// TIA Portal V17 export
// export: Created 2022-03-12T16:05:14.101526Z, ExportSetting WithDefaults, DisplayName Totally Integrated Automation Portal, DisplayVersion V17, DisplayName TIA Portal Openness, DisplayVersion V17, DisplayName TIA Portal Version Control Interface, DisplayVersion V17, DisplayName STEP 7 Professional, DisplayVersion V17, DisplayName STEP 7 Safety, DisplayVersion V17, DisplayName WinCC Advanced / Unified PC, DisplayVersion V17
FUNCTION_BLOCK "UN_01_PackML_ModuleSum"   // FB31621, LAD
TITLE = UN_01_PackML_ModuleSummation
{ S7_Optimized_Access := 'TRUE' }
AUTHOR : tech.team.motioncontrol@siemens.com
FAMILY : CPG
VERSION : 1.0
// Support: tech.team.motioncontrol@siemens.com
// Fax: +49 (0) 9131/98-1297
// stored: AutoNumber true, IsIECCheckEnabled false, IsRetainMemResEnabled false, MemoryReserve 100, SetENOAutomatically false, UDAEnableTagReadback false
   VAR
      statDummyBool { ExternalAccessible := 'False'; ExternalVisible := 'False'; ExternalWritable := 'False'} : Bool;   // dummy bool - placeholder
   END_VAR
BEGIN

REGION Network 1: UN - Reset Command
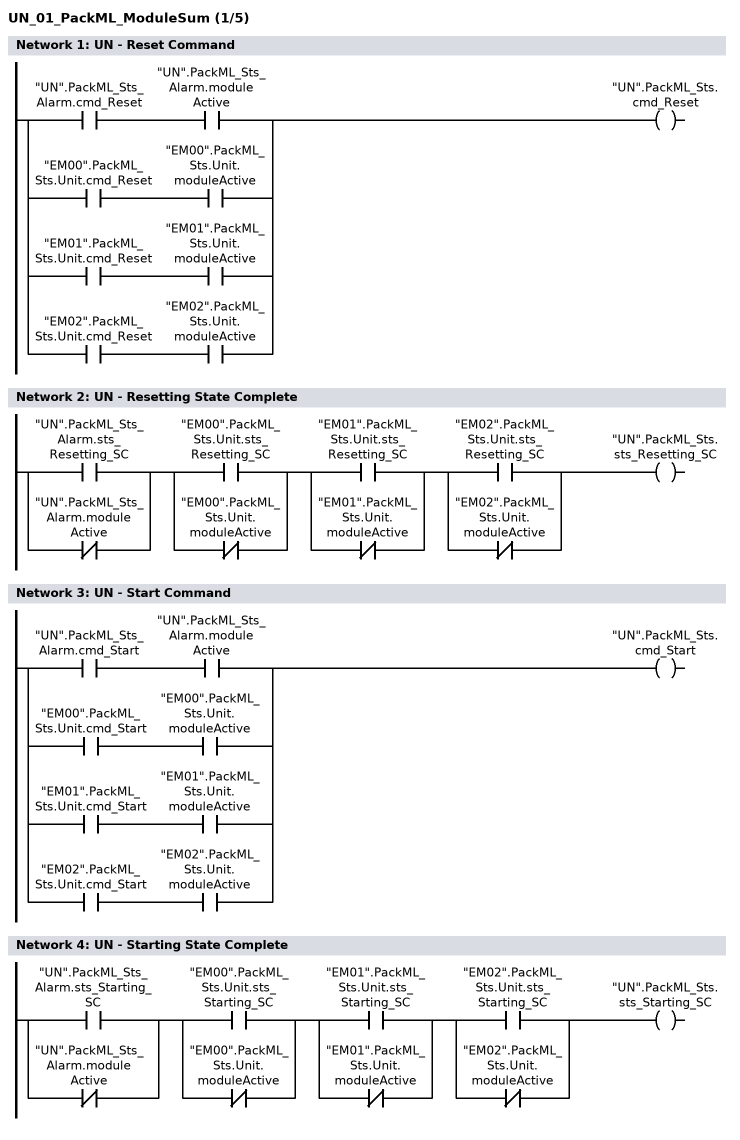
   RUNG wire#powerrail
      Contact( "UN".PackML_Sts_Alarm.cmd_Reset )
      Contact( "UN".PackML_Sts_Alarm.moduleActive )
      wire#w1
      Coil( "UN".PackML_Sts.cmd_Reset )
   END_RUNG
   RUNG wire#powerrail
      Contact( "EM00".PackML_Sts.Unit.cmd_Reset )
      Contact( "EM00".PackML_Sts.Unit.moduleActive )
   END_RUNG wire#w1
   RUNG wire#powerrail
      Contact( "EM01".PackML_Sts.Unit.cmd_Reset )
      Contact( "EM01".PackML_Sts.Unit.moduleActive )
   END_RUNG wire#w1
   RUNG wire#powerrail
      Contact( "EM02".PackML_Sts.Unit.cmd_Reset )
      Contact( "EM02".PackML_Sts.Unit.moduleActive )
   END_RUNG wire#w1
   // the same network as SCL:
   "UN".PackML_Sts.cmd_Reset := ("UN".PackML_Sts_Alarm.cmd_Reset AND "UN".PackML_Sts_Alarm.moduleActive) OR ("EM00".PackML_Sts.Unit.cmd_Reset AND "EM00".PackML_Sts.Unit.moduleActive) OR ("EM01".PackML_Sts.Unit.cmd_Reset AND "EM01".PackML_Sts.Unit.moduleActive) OR ("EM02".PackML_Sts.Unit.cmd_Reset AND "EM02".PackML_Sts.Unit.moduleActive);
END_REGION

REGION Network 2: UN - Resetting State Complete
   RUNG wire#powerrail
      Contact( "UN".PackML_Sts_Alarm.sts_Resetting_SC )
      wire#w1
      Contact( "EM00".PackML_Sts.Unit.sts_Resetting_SC )
      wire#w2
      Contact( "EM01".PackML_Sts.Unit.sts_Resetting_SC )
      wire#w3
      Contact( "EM02".PackML_Sts.Unit.sts_Resetting_SC )
      wire#w4
      Coil( "UN".PackML_Sts.sts_Resetting_SC )
   END_RUNG
   RUNG wire#powerrail
      I_Contact( "UN".PackML_Sts_Alarm.moduleActive )
   END_RUNG wire#w1
   RUNG wire#w1
      I_Contact( "EM00".PackML_Sts.Unit.moduleActive )
   END_RUNG wire#w2
   RUNG wire#w2
      I_Contact( "EM01".PackML_Sts.Unit.moduleActive )
   END_RUNG wire#w3
   RUNG wire#w3
      I_Contact( "EM02".PackML_Sts.Unit.moduleActive )
   END_RUNG wire#w4
   // the same network as SCL:
   "UN".PackML_Sts.sts_Resetting_SC := ("UN".PackML_Sts_Alarm.sts_Resetting_SC OR NOT "UN".PackML_Sts_Alarm.moduleActive) AND ("EM00".PackML_Sts.Unit.sts_Resetting_SC OR NOT "EM00".PackML_Sts.Unit.moduleActive) AND ("EM01".PackML_Sts.Unit.sts_Resetting_SC OR NOT "EM01".PackML_Sts.Unit.moduleActive) AND ("EM02".PackML_Sts.Unit.sts_Resetting_SC OR NOT "EM02".PackML_Sts.Unit.moduleActive);
END_REGION

REGION Network 3: UN - Start Command
   RUNG wire#powerrail
      Contact( "UN".PackML_Sts_Alarm.cmd_Start )
      Contact( "UN".PackML_Sts_Alarm.moduleActive )
      wire#w1
      Coil( "UN".PackML_Sts.cmd_Start )
   END_RUNG
   RUNG wire#powerrail
      Contact( "EM00".PackML_Sts.Unit.cmd_Start )
      Contact( "EM00".PackML_Sts.Unit.moduleActive )
   END_RUNG wire#w1
   RUNG wire#powerrail
      Contact( "EM01".PackML_Sts.Unit.cmd_Start )
      Contact( "EM01".PackML_Sts.Unit.moduleActive )
   END_RUNG wire#w1
   RUNG wire#powerrail
      Contact( "EM02".PackML_Sts.Unit.cmd_Start )
      Contact( "EM02".PackML_Sts.Unit.moduleActive )
   END_RUNG wire#w1
   // the same network as SCL:
   "UN".PackML_Sts.cmd_Start := ("UN".PackML_Sts_Alarm.cmd_Start AND "UN".PackML_Sts_Alarm.moduleActive) OR ("EM00".PackML_Sts.Unit.cmd_Start AND "EM00".PackML_Sts.Unit.moduleActive) OR ("EM01".PackML_Sts.Unit.cmd_Start AND "EM01".PackML_Sts.Unit.moduleActive) OR ("EM02".PackML_Sts.Unit.cmd_Start AND "EM02".PackML_Sts.Unit.moduleActive);
END_REGION

REGION Network 4: UN - Starting State Complete
   RUNG wire#powerrail
      Contact( "UN".PackML_Sts_Alarm.sts_Starting_SC )
      wire#w1
      Contact( "EM00".PackML_Sts.Unit.sts_Starting_SC )
      wire#w2
      Contact( "EM01".PackML_Sts.Unit.sts_Starting_SC )
      wire#w3
      Contact( "EM02".PackML_Sts.Unit.sts_Starting_SC )
      wire#w4
      Coil( "UN".PackML_Sts.sts_Starting_SC )
   END_RUNG
   RUNG wire#powerrail
      I_Contact( "UN".PackML_Sts_Alarm.moduleActive )
   END_RUNG wire#w1
   RUNG wire#w1
      I_Contact( "EM00".PackML_Sts.Unit.moduleActive )
   END_RUNG wire#w2
   RUNG wire#w2
      I_Contact( "EM01".PackML_Sts.Unit.moduleActive )
   END_RUNG wire#w3
   RUNG wire#w3
      I_Contact( "EM02".PackML_Sts.Unit.moduleActive )
   END_RUNG wire#w4
   // the same network as SCL:
   "UN".PackML_Sts.sts_Starting_SC := ("UN".PackML_Sts_Alarm.sts_Starting_SC OR NOT "UN".PackML_Sts_Alarm.moduleActive) AND ("EM00".PackML_Sts.Unit.sts_Starting_SC OR NOT "EM00".PackML_Sts.Unit.moduleActive) AND ("EM01".PackML_Sts.Unit.sts_Starting_SC OR NOT "EM01".PackML_Sts.Unit.moduleActive) AND ("EM02".PackML_Sts.Unit.sts_Starting_SC OR NOT "EM02".PackML_Sts.Unit.moduleActive);
END_REGION

REGION Network 5: UN - Stop Command
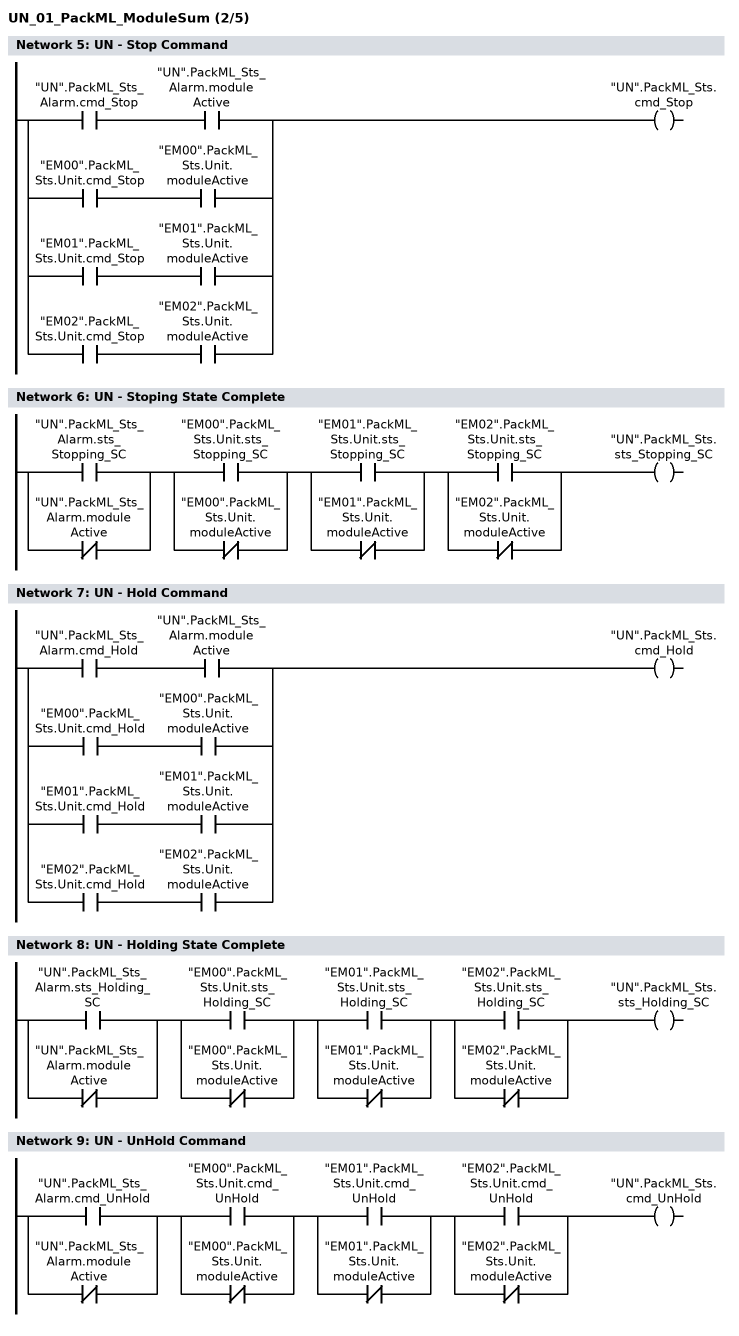
   RUNG wire#powerrail
      Contact( "UN".PackML_Sts_Alarm.cmd_Stop )
      Contact( "UN".PackML_Sts_Alarm.moduleActive )
      wire#w1
      Coil( "UN".PackML_Sts.cmd_Stop )
   END_RUNG
   RUNG wire#powerrail
      Contact( "EM00".PackML_Sts.Unit.cmd_Stop )
      Contact( "EM00".PackML_Sts.Unit.moduleActive )
   END_RUNG wire#w1
   RUNG wire#powerrail
      Contact( "EM01".PackML_Sts.Unit.cmd_Stop )
      Contact( "EM01".PackML_Sts.Unit.moduleActive )
   END_RUNG wire#w1
   RUNG wire#powerrail
      Contact( "EM02".PackML_Sts.Unit.cmd_Stop )
      Contact( "EM02".PackML_Sts.Unit.moduleActive )
   END_RUNG wire#w1
   // the same network as SCL:
   "UN".PackML_Sts.cmd_Stop := ("UN".PackML_Sts_Alarm.cmd_Stop AND "UN".PackML_Sts_Alarm.moduleActive) OR ("EM00".PackML_Sts.Unit.cmd_Stop AND "EM00".PackML_Sts.Unit.moduleActive) OR ("EM01".PackML_Sts.Unit.cmd_Stop AND "EM01".PackML_Sts.Unit.moduleActive) OR ("EM02".PackML_Sts.Unit.cmd_Stop AND "EM02".PackML_Sts.Unit.moduleActive);
END_REGION

REGION Network 6: UN - Stoping State Complete
   RUNG wire#powerrail
      Contact( "UN".PackML_Sts_Alarm.sts_Stopping_SC )
      wire#w1
      Contact( "EM00".PackML_Sts.Unit.sts_Stopping_SC )
      wire#w2
      Contact( "EM01".PackML_Sts.Unit.sts_Stopping_SC )
      wire#w3
      Contact( "EM02".PackML_Sts.Unit.sts_Stopping_SC )
      wire#w4
      Coil( "UN".PackML_Sts.sts_Stopping_SC )
   END_RUNG
   RUNG wire#powerrail
      I_Contact( "UN".PackML_Sts_Alarm.moduleActive )
   END_RUNG wire#w1
   RUNG wire#w1
      I_Contact( "EM00".PackML_Sts.Unit.moduleActive )
   END_RUNG wire#w2
   RUNG wire#w2
      I_Contact( "EM01".PackML_Sts.Unit.moduleActive )
   END_RUNG wire#w3
   RUNG wire#w3
      I_Contact( "EM02".PackML_Sts.Unit.moduleActive )
   END_RUNG wire#w4
   // the same network as SCL:
   "UN".PackML_Sts.sts_Stopping_SC := ("UN".PackML_Sts_Alarm.sts_Stopping_SC OR NOT "UN".PackML_Sts_Alarm.moduleActive) AND ("EM00".PackML_Sts.Unit.sts_Stopping_SC OR NOT "EM00".PackML_Sts.Unit.moduleActive) AND ("EM01".PackML_Sts.Unit.sts_Stopping_SC OR NOT "EM01".PackML_Sts.Unit.moduleActive) AND ("EM02".PackML_Sts.Unit.sts_Stopping_SC OR NOT "EM02".PackML_Sts.Unit.moduleActive);
END_REGION

REGION Network 7: UN - Hold Command
   RUNG wire#powerrail
      Contact( "UN".PackML_Sts_Alarm.cmd_Hold )
      Contact( "UN".PackML_Sts_Alarm.moduleActive )
      wire#w1
      Coil( "UN".PackML_Sts.cmd_Hold )
   END_RUNG
   RUNG wire#powerrail
      Contact( "EM00".PackML_Sts.Unit.cmd_Hold )
      Contact( "EM00".PackML_Sts.Unit.moduleActive )
   END_RUNG wire#w1
   RUNG wire#powerrail
      Contact( "EM01".PackML_Sts.Unit.cmd_Hold )
      Contact( "EM01".PackML_Sts.Unit.moduleActive )
   END_RUNG wire#w1
   RUNG wire#powerrail
      Contact( "EM02".PackML_Sts.Unit.cmd_Hold )
      Contact( "EM02".PackML_Sts.Unit.moduleActive )
   END_RUNG wire#w1
   // the same network as SCL:
   "UN".PackML_Sts.cmd_Hold := ("UN".PackML_Sts_Alarm.cmd_Hold AND "UN".PackML_Sts_Alarm.moduleActive) OR ("EM00".PackML_Sts.Unit.cmd_Hold AND "EM00".PackML_Sts.Unit.moduleActive) OR ("EM01".PackML_Sts.Unit.cmd_Hold AND "EM01".PackML_Sts.Unit.moduleActive) OR ("EM02".PackML_Sts.Unit.cmd_Hold AND "EM02".PackML_Sts.Unit.moduleActive);
END_REGION

REGION Network 8: UN - Holding State Complete
   RUNG wire#powerrail
      Contact( "UN".PackML_Sts_Alarm.sts_Holding_SC )
      wire#w1
      Contact( "EM00".PackML_Sts.Unit.sts_Holding_SC )
      wire#w2
      Contact( "EM01".PackML_Sts.Unit.sts_Holding_SC )
      wire#w3
      Contact( "EM02".PackML_Sts.Unit.sts_Holding_SC )
      wire#w4
      Coil( "UN".PackML_Sts.sts_Holding_SC )
   END_RUNG
   RUNG wire#powerrail
      I_Contact( "UN".PackML_Sts_Alarm.moduleActive )
   END_RUNG wire#w1
   RUNG wire#w1
      I_Contact( "EM00".PackML_Sts.Unit.moduleActive )
   END_RUNG wire#w2
   RUNG wire#w2
      I_Contact( "EM01".PackML_Sts.Unit.moduleActive )
   END_RUNG wire#w3
   RUNG wire#w3
      I_Contact( "EM02".PackML_Sts.Unit.moduleActive )
   END_RUNG wire#w4
   // the same network as SCL:
   "UN".PackML_Sts.sts_Holding_SC := ("UN".PackML_Sts_Alarm.sts_Holding_SC OR NOT "UN".PackML_Sts_Alarm.moduleActive) AND ("EM00".PackML_Sts.Unit.sts_Holding_SC OR NOT "EM00".PackML_Sts.Unit.moduleActive) AND ("EM01".PackML_Sts.Unit.sts_Holding_SC OR NOT "EM01".PackML_Sts.Unit.moduleActive) AND ("EM02".PackML_Sts.Unit.sts_Holding_SC OR NOT "EM02".PackML_Sts.Unit.moduleActive);
END_REGION

REGION Network 9: UN - UnHold Command
   RUNG wire#powerrail
      Contact( "UN".PackML_Sts_Alarm.cmd_UnHold )
      wire#w1
      Contact( "EM00".PackML_Sts.Unit.cmd_UnHold )
      wire#w2
      Contact( "EM01".PackML_Sts.Unit.cmd_UnHold )
      wire#w3
      Contact( "EM02".PackML_Sts.Unit.cmd_UnHold )
      wire#w4
      Coil( "UN".PackML_Sts.cmd_UnHold )
   END_RUNG
   RUNG wire#powerrail
      I_Contact( "UN".PackML_Sts_Alarm.moduleActive )
   END_RUNG wire#w1
   RUNG wire#w1
      I_Contact( "EM00".PackML_Sts.Unit.moduleActive )
   END_RUNG wire#w2
   RUNG wire#w2
      I_Contact( "EM01".PackML_Sts.Unit.moduleActive )
   END_RUNG wire#w3
   RUNG wire#w3
      I_Contact( "EM02".PackML_Sts.Unit.moduleActive )
   END_RUNG wire#w4
   // the same network as SCL:
   "UN".PackML_Sts.cmd_UnHold := ("UN".PackML_Sts_Alarm.cmd_UnHold OR NOT "UN".PackML_Sts_Alarm.moduleActive) AND ("EM00".PackML_Sts.Unit.cmd_UnHold OR NOT "EM00".PackML_Sts.Unit.moduleActive) AND ("EM01".PackML_Sts.Unit.cmd_UnHold OR NOT "EM01".PackML_Sts.Unit.moduleActive) AND ("EM02".PackML_Sts.Unit.cmd_UnHold OR NOT "EM02".PackML_Sts.Unit.moduleActive);
END_REGION

REGION Network 10: UN - UnHolding State Complete
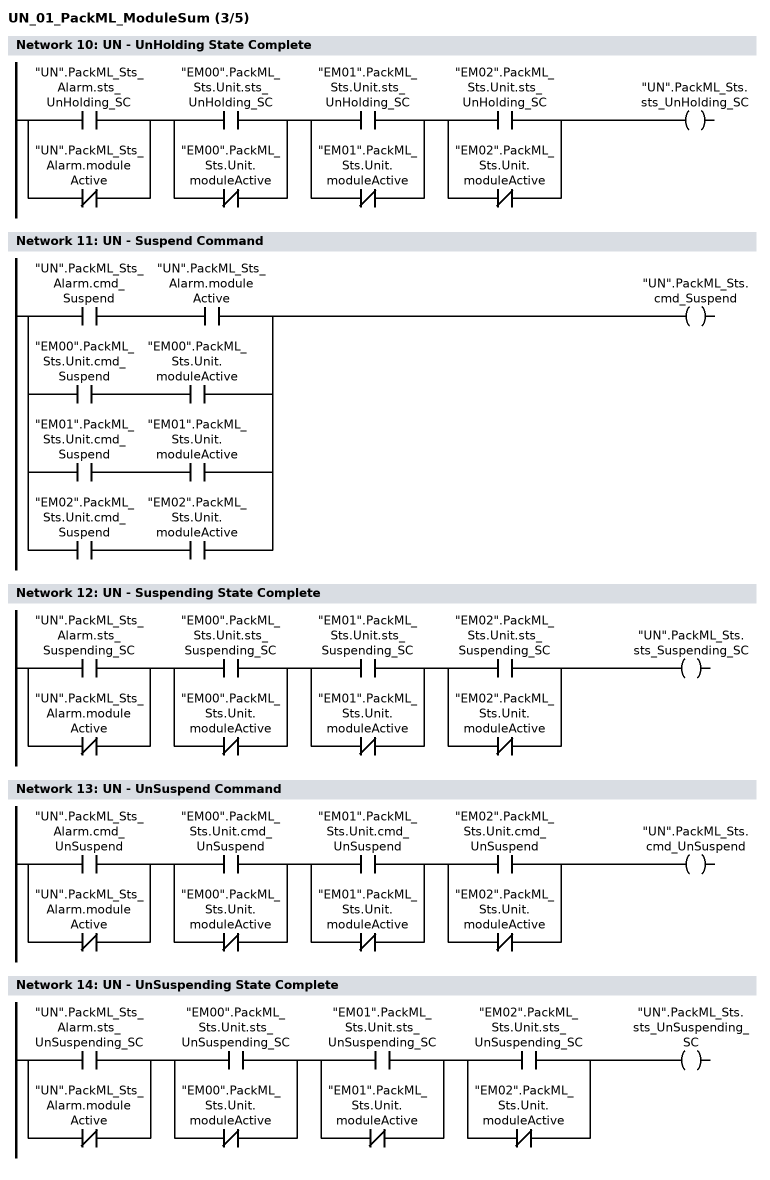
   RUNG wire#powerrail
      Contact( "UN".PackML_Sts_Alarm.sts_UnHolding_SC )
      wire#w1
      Contact( "EM00".PackML_Sts.Unit.sts_UnHolding_SC )
      wire#w2
      Contact( "EM01".PackML_Sts.Unit.sts_UnHolding_SC )
      wire#w3
      Contact( "EM02".PackML_Sts.Unit.sts_UnHolding_SC )
      wire#w4
      Coil( "UN".PackML_Sts.sts_UnHolding_SC )
   END_RUNG
   RUNG wire#powerrail
      I_Contact( "UN".PackML_Sts_Alarm.moduleActive )
   END_RUNG wire#w1
   RUNG wire#w1
      I_Contact( "EM00".PackML_Sts.Unit.moduleActive )
   END_RUNG wire#w2
   RUNG wire#w2
      I_Contact( "EM01".PackML_Sts.Unit.moduleActive )
   END_RUNG wire#w3
   RUNG wire#w3
      I_Contact( "EM02".PackML_Sts.Unit.moduleActive )
   END_RUNG wire#w4
   // the same network as SCL:
   "UN".PackML_Sts.sts_UnHolding_SC := ("UN".PackML_Sts_Alarm.sts_UnHolding_SC OR NOT "UN".PackML_Sts_Alarm.moduleActive) AND ("EM00".PackML_Sts.Unit.sts_UnHolding_SC OR NOT "EM00".PackML_Sts.Unit.moduleActive) AND ("EM01".PackML_Sts.Unit.sts_UnHolding_SC OR NOT "EM01".PackML_Sts.Unit.moduleActive) AND ("EM02".PackML_Sts.Unit.sts_UnHolding_SC OR NOT "EM02".PackML_Sts.Unit.moduleActive);
END_REGION

REGION Network 11: UN - Suspend Command
   RUNG wire#powerrail
      Contact( "UN".PackML_Sts_Alarm.cmd_Suspend )
      Contact( "UN".PackML_Sts_Alarm.moduleActive )
      wire#w1
      Coil( "UN".PackML_Sts.cmd_Suspend )
   END_RUNG
   RUNG wire#powerrail
      Contact( "EM00".PackML_Sts.Unit.cmd_Suspend )
      Contact( "EM00".PackML_Sts.Unit.moduleActive )
   END_RUNG wire#w1
   RUNG wire#powerrail
      Contact( "EM01".PackML_Sts.Unit.cmd_Suspend )
      Contact( "EM01".PackML_Sts.Unit.moduleActive )
   END_RUNG wire#w1
   RUNG wire#powerrail
      Contact( "EM02".PackML_Sts.Unit.cmd_Suspend )
      Contact( "EM02".PackML_Sts.Unit.moduleActive )
   END_RUNG wire#w1
   // the same network as SCL:
   "UN".PackML_Sts.cmd_Suspend := ("UN".PackML_Sts_Alarm.cmd_Suspend AND "UN".PackML_Sts_Alarm.moduleActive) OR ("EM00".PackML_Sts.Unit.cmd_Suspend AND "EM00".PackML_Sts.Unit.moduleActive) OR ("EM01".PackML_Sts.Unit.cmd_Suspend AND "EM01".PackML_Sts.Unit.moduleActive) OR ("EM02".PackML_Sts.Unit.cmd_Suspend AND "EM02".PackML_Sts.Unit.moduleActive);
END_REGION

REGION Network 12: UN - Suspending State Complete
   RUNG wire#powerrail
      Contact( "UN".PackML_Sts_Alarm.sts_Suspending_SC )
      wire#w1
      Contact( "EM00".PackML_Sts.Unit.sts_Suspending_SC )
      wire#w2
      Contact( "EM01".PackML_Sts.Unit.sts_Suspending_SC )
      wire#w3
      Contact( "EM02".PackML_Sts.Unit.sts_Suspending_SC )
      wire#w4
      Coil( "UN".PackML_Sts.sts_Suspending_SC )
   END_RUNG
   RUNG wire#powerrail
      I_Contact( "UN".PackML_Sts_Alarm.moduleActive )
   END_RUNG wire#w1
   RUNG wire#w1
      I_Contact( "EM00".PackML_Sts.Unit.moduleActive )
   END_RUNG wire#w2
   RUNG wire#w2
      I_Contact( "EM01".PackML_Sts.Unit.moduleActive )
   END_RUNG wire#w3
   RUNG wire#w3
      I_Contact( "EM02".PackML_Sts.Unit.moduleActive )
   END_RUNG wire#w4
   // the same network as SCL:
   "UN".PackML_Sts.sts_Suspending_SC := ("UN".PackML_Sts_Alarm.sts_Suspending_SC OR NOT "UN".PackML_Sts_Alarm.moduleActive) AND ("EM00".PackML_Sts.Unit.sts_Suspending_SC OR NOT "EM00".PackML_Sts.Unit.moduleActive) AND ("EM01".PackML_Sts.Unit.sts_Suspending_SC OR NOT "EM01".PackML_Sts.Unit.moduleActive) AND ("EM02".PackML_Sts.Unit.sts_Suspending_SC OR NOT "EM02".PackML_Sts.Unit.moduleActive);
END_REGION

REGION Network 13: UN - UnSuspend Command
   RUNG wire#powerrail
      Contact( "UN".PackML_Sts_Alarm.cmd_UnSuspend )
      wire#w1
      Contact( "EM00".PackML_Sts.Unit.cmd_UnSuspend )
      wire#w2
      Contact( "EM01".PackML_Sts.Unit.cmd_UnSuspend )
      wire#w3
      Contact( "EM02".PackML_Sts.Unit.cmd_UnSuspend )
      wire#w4
      Coil( "UN".PackML_Sts.cmd_UnSuspend )
   END_RUNG
   RUNG wire#powerrail
      I_Contact( "UN".PackML_Sts_Alarm.moduleActive )
   END_RUNG wire#w1
   RUNG wire#w1
      I_Contact( "EM00".PackML_Sts.Unit.moduleActive )
   END_RUNG wire#w2
   RUNG wire#w2
      I_Contact( "EM01".PackML_Sts.Unit.moduleActive )
   END_RUNG wire#w3
   RUNG wire#w3
      I_Contact( "EM02".PackML_Sts.Unit.moduleActive )
   END_RUNG wire#w4
   // the same network as SCL:
   "UN".PackML_Sts.cmd_UnSuspend := ("UN".PackML_Sts_Alarm.cmd_UnSuspend OR NOT "UN".PackML_Sts_Alarm.moduleActive) AND ("EM00".PackML_Sts.Unit.cmd_UnSuspend OR NOT "EM00".PackML_Sts.Unit.moduleActive) AND ("EM01".PackML_Sts.Unit.cmd_UnSuspend OR NOT "EM01".PackML_Sts.Unit.moduleActive) AND ("EM02".PackML_Sts.Unit.cmd_UnSuspend OR NOT "EM02".PackML_Sts.Unit.moduleActive);
END_REGION

REGION Network 14: UN - UnSuspending State Complete
   RUNG wire#powerrail
      Contact( "UN".PackML_Sts_Alarm.sts_UnSuspending_SC )
      wire#w1
      Contact( "EM00".PackML_Sts.Unit.sts_UnSuspending_SC )
      wire#w2
      Contact( "EM01".PackML_Sts.Unit.sts_UnSuspending_SC )
      wire#w3
      Contact( "EM02".PackML_Sts.Unit.sts_UnSuspending_SC )
      wire#w4
      Coil( "UN".PackML_Sts.sts_UnSuspending_SC )
   END_RUNG
   RUNG wire#powerrail
      I_Contact( "UN".PackML_Sts_Alarm.moduleActive )
   END_RUNG wire#w1
   RUNG wire#w1
      I_Contact( "EM00".PackML_Sts.Unit.moduleActive )
   END_RUNG wire#w2
   RUNG wire#w2
      I_Contact( "EM01".PackML_Sts.Unit.moduleActive )
   END_RUNG wire#w3
   RUNG wire#w3
      I_Contact( "EM02".PackML_Sts.Unit.moduleActive )
   END_RUNG wire#w4
   // the same network as SCL:
   "UN".PackML_Sts.sts_UnSuspending_SC := ("UN".PackML_Sts_Alarm.sts_UnSuspending_SC OR NOT "UN".PackML_Sts_Alarm.moduleActive) AND ("EM00".PackML_Sts.Unit.sts_UnSuspending_SC OR NOT "EM00".PackML_Sts.Unit.moduleActive) AND ("EM01".PackML_Sts.Unit.sts_UnSuspending_SC OR NOT "EM01".PackML_Sts.Unit.moduleActive) AND ("EM02".PackML_Sts.Unit.sts_UnSuspending_SC OR NOT "EM02".PackML_Sts.Unit.moduleActive);
END_REGION

REGION Network 15: UN - Abort Command
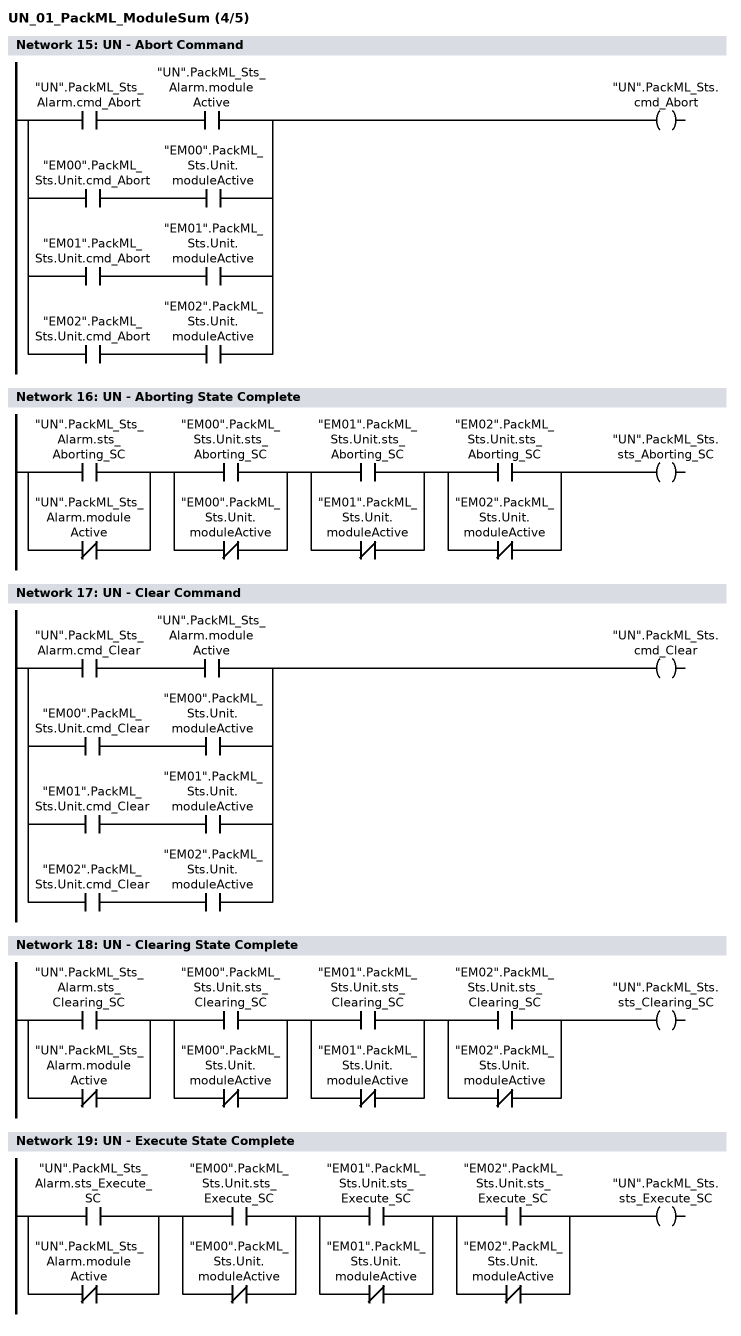
   RUNG wire#powerrail
      Contact( "UN".PackML_Sts_Alarm.cmd_Abort )
      Contact( "UN".PackML_Sts_Alarm.moduleActive )
      wire#w1
      Coil( "UN".PackML_Sts.cmd_Abort )
   END_RUNG
   RUNG wire#powerrail
      Contact( "EM00".PackML_Sts.Unit.cmd_Abort )
      Contact( "EM00".PackML_Sts.Unit.moduleActive )
   END_RUNG wire#w1
   RUNG wire#powerrail
      Contact( "EM01".PackML_Sts.Unit.cmd_Abort )
      Contact( "EM01".PackML_Sts.Unit.moduleActive )
   END_RUNG wire#w1
   RUNG wire#powerrail
      Contact( "EM02".PackML_Sts.Unit.cmd_Abort )
      Contact( "EM02".PackML_Sts.Unit.moduleActive )
   END_RUNG wire#w1
   // the same network as SCL:
   "UN".PackML_Sts.cmd_Abort := ("UN".PackML_Sts_Alarm.cmd_Abort AND "UN".PackML_Sts_Alarm.moduleActive) OR ("EM00".PackML_Sts.Unit.cmd_Abort AND "EM00".PackML_Sts.Unit.moduleActive) OR ("EM01".PackML_Sts.Unit.cmd_Abort AND "EM01".PackML_Sts.Unit.moduleActive) OR ("EM02".PackML_Sts.Unit.cmd_Abort AND "EM02".PackML_Sts.Unit.moduleActive);
END_REGION

REGION Network 16: UN - Aborting State Complete
   RUNG wire#powerrail
      Contact( "UN".PackML_Sts_Alarm.sts_Aborting_SC )
      wire#w1
      Contact( "EM00".PackML_Sts.Unit.sts_Aborting_SC )
      wire#w2
      Contact( "EM01".PackML_Sts.Unit.sts_Aborting_SC )
      wire#w3
      Contact( "EM02".PackML_Sts.Unit.sts_Aborting_SC )
      wire#w4
      Coil( "UN".PackML_Sts.sts_Aborting_SC )
   END_RUNG
   RUNG wire#powerrail
      I_Contact( "UN".PackML_Sts_Alarm.moduleActive )
   END_RUNG wire#w1
   RUNG wire#w1
      I_Contact( "EM00".PackML_Sts.Unit.moduleActive )
   END_RUNG wire#w2
   RUNG wire#w2
      I_Contact( "EM01".PackML_Sts.Unit.moduleActive )
   END_RUNG wire#w3
   RUNG wire#w3
      I_Contact( "EM02".PackML_Sts.Unit.moduleActive )
   END_RUNG wire#w4
   // the same network as SCL:
   "UN".PackML_Sts.sts_Aborting_SC := ("UN".PackML_Sts_Alarm.sts_Aborting_SC OR NOT "UN".PackML_Sts_Alarm.moduleActive) AND ("EM00".PackML_Sts.Unit.sts_Aborting_SC OR NOT "EM00".PackML_Sts.Unit.moduleActive) AND ("EM01".PackML_Sts.Unit.sts_Aborting_SC OR NOT "EM01".PackML_Sts.Unit.moduleActive) AND ("EM02".PackML_Sts.Unit.sts_Aborting_SC OR NOT "EM02".PackML_Sts.Unit.moduleActive);
END_REGION

REGION Network 17: UN - Clear Command
   RUNG wire#powerrail
      Contact( "UN".PackML_Sts_Alarm.cmd_Clear )
      Contact( "UN".PackML_Sts_Alarm.moduleActive )
      wire#w1
      Coil( "UN".PackML_Sts.cmd_Clear )
   END_RUNG
   RUNG wire#powerrail
      Contact( "EM00".PackML_Sts.Unit.cmd_Clear )
      Contact( "EM00".PackML_Sts.Unit.moduleActive )
   END_RUNG wire#w1
   RUNG wire#powerrail
      Contact( "EM01".PackML_Sts.Unit.cmd_Clear )
      Contact( "EM01".PackML_Sts.Unit.moduleActive )
   END_RUNG wire#w1
   RUNG wire#powerrail
      Contact( "EM02".PackML_Sts.Unit.cmd_Clear )
      Contact( "EM02".PackML_Sts.Unit.moduleActive )
   END_RUNG wire#w1
   // the same network as SCL:
   "UN".PackML_Sts.cmd_Clear := ("UN".PackML_Sts_Alarm.cmd_Clear AND "UN".PackML_Sts_Alarm.moduleActive) OR ("EM00".PackML_Sts.Unit.cmd_Clear AND "EM00".PackML_Sts.Unit.moduleActive) OR ("EM01".PackML_Sts.Unit.cmd_Clear AND "EM01".PackML_Sts.Unit.moduleActive) OR ("EM02".PackML_Sts.Unit.cmd_Clear AND "EM02".PackML_Sts.Unit.moduleActive);
END_REGION

REGION Network 18: UN - Clearing State Complete
   RUNG wire#powerrail
      Contact( "UN".PackML_Sts_Alarm.sts_Clearing_SC )
      wire#w1
      Contact( "EM00".PackML_Sts.Unit.sts_Clearing_SC )
      wire#w2
      Contact( "EM01".PackML_Sts.Unit.sts_Clearing_SC )
      wire#w3
      Contact( "EM02".PackML_Sts.Unit.sts_Clearing_SC )
      wire#w4
      Coil( "UN".PackML_Sts.sts_Clearing_SC )
   END_RUNG
   RUNG wire#powerrail
      I_Contact( "UN".PackML_Sts_Alarm.moduleActive )
   END_RUNG wire#w1
   RUNG wire#w1
      I_Contact( "EM00".PackML_Sts.Unit.moduleActive )
   END_RUNG wire#w2
   RUNG wire#w2
      I_Contact( "EM01".PackML_Sts.Unit.moduleActive )
   END_RUNG wire#w3
   RUNG wire#w3
      I_Contact( "EM02".PackML_Sts.Unit.moduleActive )
   END_RUNG wire#w4
   // the same network as SCL:
   "UN".PackML_Sts.sts_Clearing_SC := ("UN".PackML_Sts_Alarm.sts_Clearing_SC OR NOT "UN".PackML_Sts_Alarm.moduleActive) AND ("EM00".PackML_Sts.Unit.sts_Clearing_SC OR NOT "EM00".PackML_Sts.Unit.moduleActive) AND ("EM01".PackML_Sts.Unit.sts_Clearing_SC OR NOT "EM01".PackML_Sts.Unit.moduleActive) AND ("EM02".PackML_Sts.Unit.sts_Clearing_SC OR NOT "EM02".PackML_Sts.Unit.moduleActive);
END_REGION

REGION Network 19: UN - Execute State Complete
   RUNG wire#powerrail
      Contact( "UN".PackML_Sts_Alarm.sts_Execute_SC )
      wire#w1
      Contact( "EM00".PackML_Sts.Unit.sts_Execute_SC )
      wire#w2
      Contact( "EM01".PackML_Sts.Unit.sts_Execute_SC )
      wire#w3
      Contact( "EM02".PackML_Sts.Unit.sts_Execute_SC )
      wire#w4
      Coil( "UN".PackML_Sts.sts_Execute_SC )
   END_RUNG
   RUNG wire#powerrail
      I_Contact( "UN".PackML_Sts_Alarm.moduleActive )
   END_RUNG wire#w1
   RUNG wire#w1
      I_Contact( "EM00".PackML_Sts.Unit.moduleActive )
   END_RUNG wire#w2
   RUNG wire#w2
      I_Contact( "EM01".PackML_Sts.Unit.moduleActive )
   END_RUNG wire#w3
   RUNG wire#w3
      I_Contact( "EM02".PackML_Sts.Unit.moduleActive )
   END_RUNG wire#w4
   // the same network as SCL:
   "UN".PackML_Sts.sts_Execute_SC := ("UN".PackML_Sts_Alarm.sts_Execute_SC OR NOT "UN".PackML_Sts_Alarm.moduleActive) AND ("EM00".PackML_Sts.Unit.sts_Execute_SC OR NOT "EM00".PackML_Sts.Unit.moduleActive) AND ("EM01".PackML_Sts.Unit.sts_Execute_SC OR NOT "EM01".PackML_Sts.Unit.moduleActive) AND ("EM02".PackML_Sts.Unit.sts_Execute_SC OR NOT "EM02".PackML_Sts.Unit.moduleActive);
END_REGION

REGION Network 20: UN - Completing State Complete
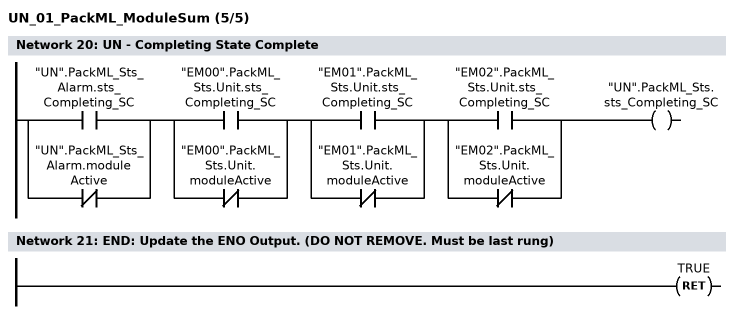
   RUNG wire#powerrail
      Contact( "UN".PackML_Sts_Alarm.sts_Completing_SC )
      wire#w1
      Contact( "EM00".PackML_Sts.Unit.sts_Completing_SC )
      wire#w2
      Contact( "EM01".PackML_Sts.Unit.sts_Completing_SC )
      wire#w3
      Contact( "EM02".PackML_Sts.Unit.sts_Completing_SC )
      wire#w4
      Coil( "UN".PackML_Sts.sts_Completing_SC )
   END_RUNG
   RUNG wire#powerrail
      I_Contact( "UN".PackML_Sts_Alarm.moduleActive )
   END_RUNG wire#w1
   RUNG wire#w1
      I_Contact( "EM00".PackML_Sts.Unit.moduleActive )
   END_RUNG wire#w2
   RUNG wire#w2
      I_Contact( "EM01".PackML_Sts.Unit.moduleActive )
   END_RUNG wire#w3
   RUNG wire#w3
      I_Contact( "EM02".PackML_Sts.Unit.moduleActive )
   END_RUNG wire#w4
   // the same network as SCL:
   "UN".PackML_Sts.sts_Completing_SC := ("UN".PackML_Sts_Alarm.sts_Completing_SC OR NOT "UN".PackML_Sts_Alarm.moduleActive) AND ("EM00".PackML_Sts.Unit.sts_Completing_SC OR NOT "EM00".PackML_Sts.Unit.moduleActive) AND ("EM01".PackML_Sts.Unit.sts_Completing_SC OR NOT "EM01".PackML_Sts.Unit.moduleActive) AND ("EM02".PackML_Sts.Unit.sts_Completing_SC OR NOT "EM02".PackML_Sts.Unit.moduleActive);
END_REGION

REGION Network 21: END: Update the ENO Output. (DO NOT REMOVE. Must be last rung)
   RUNG wire#powerrail
      ReturnCoil( TRUE )
   END_RUNG
   // the same network as SCL:
   ENO := TRUE;
   RETURN;
END_REGION
END_FUNCTION_BLOCK
